// TIA Portal V19 export
TYPE "C501_STU_TME_TYPIC"
   STRUCT
      VGV_L { ExternalAccessible := 'False'; ExternalVisible := 'False'; ExternalWritable := 'False'} : USInt;   // Vrijgave detectie temperatuur te laag
   END_STRUCT;
END_TYPE
